// TwinCAT 3 PLC project Untitled1
// ProgramVersion: 3.1.4023.0
// libraries:
//   Tc2_Standard, * (Beckhoff Automation GmbH)
//   Tc2_System, * (Beckhoff Automation GmbH)
//   Tc3_Module, * (Beckhoff Automation GmbH)
// project tree:
//   / PlcTask.TcTTO
//   POUs/ MAIN.TcPOU
// real-time tasks:
//   TASK PlcTask: cycle T#10ms, priority 20, ADS port 350
// I/O:
//   DEVICE Device 1 (EtherCAT Automation Protocol), AmsNetId 5.79.69.158.2.1
//     Box 1 (Subscriber)
// variable links:
//   Untitled1/Untitled1 Instance <-> Device 1 (EtherCAT Automation Protocol)/Box 1 (Subscriber)
//     PlcTask Inputs/MAIN.nIndex <-> Pub-Var 1/Inputs/VarData
//     PlcTask Inputs/MAIN.sText <-> Pub-Var 2/Inputs/VarData

CONFIGURATION Untitled1
    RESOURCE PLC ON TwinCAT3
        TASK PlcTask(INTERVAL := T#10ms, PRIORITY := 20);
        PROGRAM MAIN WITH PlcTask : MAIN;
    END_RESOURCE
END_CONFIGURATION

// ---- POUs/MAIN.TcPOU
PROGRAM MAIN
VAR
	nIndex AT %I*		:	DINT;
	sText AT %I*		:	T_MaxString;
	nLen				:	DINT;
END_VAR

nlen := len(sText);

END_PROGRAM
